PROGRAM prgComEffIO
VAR
	fbCom		: FB_MqttCommunicator_v3;

END_VAR

fbCom(
	bConnect:= TRUE, 
	strAuthkey := 'DEV01673741737',
	sUserName:= '42cf3b23-700d-4275-a072-1301ce2666ee' , 		
	sUserPassword:= 'abe4fa5d-8e50-48f0-873c-207b5a84d6b6',
	eSavePositionCertificate:= eSavePositionOnPLC.ePostionC, 
	bConnected=> , 
	bError=> , 
	hrErrorCode=> , 
	eConnectionState=> , 
	eErrorMessage_Out=> );

END_PROGRAM

(* stored: Version 1.1.0.1, ProductVersion 3.1.4024.12
   POU prgComEffIO: Id {f69e1176-2641-4928-b934-4378d8a11b2c}, SpecialFunc None *)
